FUNCTION_BLOCK AQ_MERGE_2 (* Fan-In: Merges 2 AQ into 1 AQ adapter *)
  (* Standard: 61499-2; Description: Copyright (c) 2026 Meisterschulen am Ostbahnhof SPDX-License-Identifier: EPL-2.0 *)
  (* Version 1.0, 2026-05-16, Franz Höpfinger, Meisterschulen am Ostbahnhof, Initial Version *)
  PACKAGE adapter::events::unidirectional;
  IMPORT eclipse4diac::core::GenericClassName;
  {SET_ATTRIBUTE(eclipse4diac::core::GenericClassName, 'GEN_AQ_MERGE')}
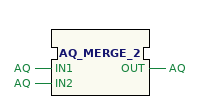
  SOCKETS
    IN1 : adapter::types::unidirectional::AQ; (* Input 1 *)
    IN2 : adapter::types::unidirectional::AQ; (* Input 2 *)
  END_SOCKETS
  PLUGS
    OUT : adapter::types::unidirectional::AQ; (* Output *)
  END_PLUGS
END_FUNCTION_BLOCK
